Staubli VAL3: HMI.pgx

program HMI()
begin
  //This routine is to is HMI to re-teach points
  call hmi_keyinmain()
end
